{attribute 'linkalways'} 
{attribute 'no_explicit_call' := 'This FB is a CLASS and must be accessed using methods or properties'}
{attribute 'enable_dynamic_creation'}
FUNCTION_BLOCK AlarmAddedEvent EXTENDS Disposable IMPLEMENTS I_AlarmAddedEvent
VAR
	_target : I_Alarm;
END_VAR

METHOD FB_init : BOOL
VAR_INPUT
	bInitRetains : BOOL; // if TRUE, the retain variables are initialized (warm start / cold start)
	bInCopyCode : BOOL;  // if TRUE, the instance afterwards gets moved into the copy code (online change)
	Target : I_Alarm;
END_VAR
This^._target := Target;
END_METHOD

PROPERTY PUBLIC Target : I_Alarm
GET
Target := _target;
END_GET
END_PROPERTY

END_FUNCTION_BLOCK

(* stored: Version 1.1.0.1, ProductVersion 3.1.4024.12
   POU AlarmAddedEvent: Id {8019204d-c3b6-02ab-1b82-98a7f9ec0627}, SpecialFunc None
   Folder Constructor: Id {90613c27-7863-0944-16c8-c6b17e85f340}
   Method FB_init: Id {0483faaf-3347-08cb-01f4-44ab7fbce7f8}
   Property Target: Id {76c0f6be-146d-011d-2992-c8ae2e9400cf}
   Get Get: Id {145585c8-2f5a-01db-04bb-0cb34ba4def4} *)
